Universal Robots URScript: script_ur3e.urscript

def ur3e_dibujar():
  textmsg("=== UR3e: inicio del programa ===")
  q_home = get_actual_joint_positions()
  textmsg("UR3e HOME guardado")
  # === Ir al origen calibrado: UR3e ===
  textmsg("UR3e - yendo al origen calibrado")
  x0 = -0.52777
  y0 = -0.01601
  z_mesa = 0.00821
  rx = 1.34600
  ry = 2.83900
  rz = 0.00000
  # Primero se acerca por arriba; nunca va directamente a la Z baja.
  movel(p[x0, y0, z_mesa+0.06000, rx, ry, rz], a=0.03, v=0.05)
  sleep(0.3)
  # === Detección única de superficie por fuerza: UR3e ===
  textmsg("UR3e - Detectando superficie una sola vez...")
  zero_ftsensor()
  sleep(0.5)
  i_f = 0
  while (force() < 2.000 and i_f < 2000):
    speedl([0, 0, -0.00800, 0, 0, 0], 0.25, 0.02)
    i_f = i_f + 1
  end
  stopl(3.0)
  sleep(0.2)
  if (i_f >= 2000):
    popup("UR3e: No se detectó superficie. Revisa posición inicial y F_UMBRAL.", error=True)
    halt
  end
  z_contacto = get_actual_tcp_pose()[2]
  z_dibujo = z_contacto + 0.00150
  textmsg("UR3e - z_contacto=", z_contacto)
  textmsg("UR3e - z_dibujo=", z_dibujo)
  movel(p[x0, y0, z_dibujo+0.02500, rx, ry, rz], a=0.03, v=0.04)
  sleep(0.2)
  # === Dibujo - UR3e - 3 trazos ===

  # --- Trazo 1 / 3 ---
  textmsg("UR3e - Trazo 1 de 3")
  movel(p[x0+-0.00248, y0+0.02956, z_dibujo+0.02500, rx, ry, rz], a=0.03, v=0.04)
  movel(p[x0+-0.00248, y0+0.02956, z_dibujo, rx, ry, rz], a=0.006, v=0.002)
  movel(p[x0+-0.00217, y0+0.02987, z_dibujo, rx, ry, rz], a=0.008, v=0.025, r=0.0002)
  movel(p[x0+0.00186, y0+0.02987, z_dibujo, rx, ry, rz], a=0.008, v=0.025, r=0.0002)
  movel(p[x0+0.00495, y0+0.02894, z_dibujo, rx, ry, rz], a=0.008, v=0.025, r=0.0002)
  movel(p[x0+0.00805, y0+0.02708, z_dibujo, rx, ry, rz], a=0.008, v=0.025, r=0.0002)
  movel(p[x0+0.00990, y0+0.02523, z_dibujo, rx, ry, rz], a=0.008, v=0.025, r=0.0002)
  movel(p[x0+0.01114, y0+0.02306, z_dibujo, rx, ry, rz], a=0.008, v=0.025, r=0.0002)
  movel(p[x0+0.01176, y0+0.02089, z_dibujo, rx, ry, rz], a=0.008, v=0.025, r=0.0002)
  movel(p[x0+0.01176, y0+0.01811, z_dibujo, rx, ry, rz], a=0.008, v=0.025, r=0.0002)
  movel(p[x0+0.01021, y0+0.01439, z_dibujo, rx, ry, rz], a=0.008, v=0.025, r=0.0002)
  movel(p[x0+0.00619, y0+0.00913, z_dibujo, rx, ry, rz], a=0.008, v=0.025, r=0.0002)
  movel(p[x0+0.00526, y0+0.00913, z_dibujo, rx, ry, rz], a=0.008, v=0.025, r=0.0002)
  movel(p[x0+0.00433, y0+0.00975, z_dibujo, rx, ry, rz], a=0.008, v=0.025, r=0.0002)
  movel(p[x0+0.00217, y0+0.01037, z_dibujo, rx, ry, rz], a=0.008, v=0.025, r=0.0002)
  movel(p[x0+-0.00217, y0+0.01037, z_dibujo, rx, ry, rz], a=0.008, v=0.025, r=0.0002)
  movel(p[x0+-0.00248, y0+0.01006, z_dibujo, rx, ry, rz], a=0.008, v=0.025, r=0.0002)
  movel(p[x0+-0.00464, y0+0.00975, z_dibujo, rx, ry, rz], a=0.008, v=0.025, r=0.0002)
  movel(p[x0+-0.00557, y0+0.00913, z_dibujo, rx, ry, rz], a=0.008, v=0.025, r=0.0002)
  movel(p[x0+-0.00650, y0+0.00913, z_dibujo, rx, ry, rz], a=0.008, v=0.025, r=0.0002)
  movel(p[x0+-0.01021, y0+0.01408, z_dibujo, rx, ry, rz], a=0.008, v=0.025, r=0.0002)
  movel(p[x0+-0.01145, y0+0.01625, z_dibujo, rx, ry, rz], a=0.008, v=0.025, r=0.0002)
  movel(p[x0+-0.01207, y0+0.01842, z_dibujo, rx, ry, rz], a=0.008, v=0.025, r=0.0002)
  movel(p[x0+-0.01207, y0+0.02058, z_dibujo, rx, ry, rz], a=0.008, v=0.025, r=0.0002)
  movel(p[x0+-0.01114, y0+0.02368, z_dibujo, rx, ry, rz], a=0.008, v=0.025, r=0.0002)
  movel(p[x0+-0.00990, y0+0.02554, z_dibujo, rx, ry, rz], a=0.008, v=0.025, r=0.0002)
  movel(p[x0+-0.00743, y0+0.02770, z_dibujo, rx, ry, rz], a=0.008, v=0.025, r=0.0002)
  movel(p[x0+-0.00526, y0+0.02894, z_dibujo, rx, ry, rz], a=0.008, v=0.025, r=0.0002)
  movel(p[x0+-0.00279, y0+0.02956, z_dibujo, rx, ry, rz], a=0.008, v=0.025, r=0.0002)
  movel(p[x0+-0.00279, y0+0.02956, z_dibujo+0.02500, rx, ry, rz], a=0.03, v=0.04)

  # --- Trazo 2 / 3 ---
  textmsg("UR3e - Trazo 2 de 3")
  movel(p[x0+0.01052, y0+-0.00696, z_dibujo+0.02500, rx, ry, rz], a=0.03, v=0.04)
  movel(p[x0+0.01052, y0+-0.00696, z_dibujo, rx, ry, rz], a=0.006, v=0.002)
  movel(p[x0+0.01083, y0+-0.00665, z_dibujo, rx, ry, rz], a=0.008, v=0.025, r=0.0002)
  movel(p[x0+0.01238, y0+-0.00665, z_dibujo, rx, ry, rz], a=0.008, v=0.025, r=0.0002)
  movel(p[x0+0.01640, y0+-0.00820, z_dibujo, rx, ry, rz], a=0.008, v=0.025, r=0.0002)
  movel(p[x0+0.01733, y0+-0.00820, z_dibujo, rx, ry, rz], a=0.008, v=0.025, r=0.0002)
  movel(p[x0+0.01919, y0+-0.00913, z_dibujo, rx, ry, rz], a=0.008, v=0.025, r=0.0002)
  movel(p[x0+0.02074, y0+-0.01037, z_dibujo, rx, ry, rz], a=0.008, v=0.025, r=0.0002)
  movel(p[x0+0.02229, y0+-0.01223, z_dibujo, rx, ry, rz], a=0.008, v=0.025, r=0.0002)
  movel(p[x0+0.02321, y0+-0.01408, z_dibujo, rx, ry, rz], a=0.008, v=0.025, r=0.0002)
  movel(p[x0+0.02352, y0+-0.01656, z_dibujo, rx, ry, rz], a=0.008, v=0.025, r=0.0002)
  movel(p[x0+0.02383, y0+-0.01687, z_dibujo, rx, ry, rz], a=0.008, v=0.025, r=0.0002)
  movel(p[x0+0.02321, y0+-0.02058, z_dibujo, rx, ry, rz], a=0.008, v=0.025, r=0.0002)
  movel(p[x0+0.02136, y0+-0.02399, z_dibujo, rx, ry, rz], a=0.008, v=0.025, r=0.0002)
  movel(p[x0+0.01857, y0+-0.02677, z_dibujo, rx, ry, rz], a=0.008, v=0.025, r=0.0002)
  movel(p[x0+0.01671, y0+-0.02801, z_dibujo, rx, ry, rz], a=0.008, v=0.025, r=0.0002)
  movel(p[x0+0.01207, y0+-0.02956, z_dibujo, rx, ry, rz], a=0.008, v=0.025, r=0.0002)
  movel(p[x0+0.00929, y0+-0.02956, z_dibujo, rx, ry, rz], a=0.008, v=0.025, r=0.0002)
  movel(p[x0+0.00526, y0+-0.02801, z_dibujo, rx, ry, rz], a=0.008, v=0.025, r=0.0002)
  movel(p[x0+0.00248, y0+-0.02523, z_dibujo, rx, ry, rz], a=0.008, v=0.025, r=0.0002)
  movel(p[x0+0.00093, y0+-0.02151, z_dibujo, rx, ry, rz], a=0.008, v=0.025, r=0.0002)
  movel(p[x0+0.00093, y0+-0.01377, z_dibujo, rx, ry, rz], a=0.008, v=0.025, r=0.0002)
  movel(p[x0+0.00124, y0+-0.01346, z_dibujo, rx, ry, rz], a=0.008, v=0.025, r=0.0002)
  movel(p[x0+0.00433, y0+-0.01285, z_dibujo, rx, ry, rz], a=0.008, v=0.025, r=0.0002)
  movel(p[x0+0.00712, y0+-0.01130, z_dibujo, rx, ry, rz], a=0.008, v=0.025, r=0.0002)
  movel(p[x0+0.00960, y0+-0.00882, z_dibujo, rx, ry, rz], a=0.008, v=0.025, r=0.0002)
  movel(p[x0+0.01052, y0+-0.00727, z_dibujo, rx, ry, rz], a=0.008, v=0.025, r=0.0002)
  movel(p[x0+0.01052, y0+-0.00727, z_dibujo+0.02500, rx, ry, rz], a=0.03, v=0.04)

  # --- Trazo 3 / 3 ---
  textmsg("UR3e - Trazo 3 de 3")
  movel(p[x0+-0.00186, y0+0.00820, z_dibujo+0.02500, rx, ry, rz], a=0.03, v=0.04)
  movel(p[x0+-0.00186, y0+0.00820, z_dibujo, rx, ry, rz], a=0.006, v=0.002)
  movel(p[x0+-0.00155, y0+0.00851, z_dibujo, rx, ry, rz], a=0.008, v=0.025, r=0.0002)
  movel(p[x0+0.00124, y0+0.00851, z_dibujo, rx, ry, rz], a=0.008, v=0.025, r=0.0002)
  movel(p[x0+0.00526, y0+0.00696, z_dibujo, rx, ry, rz], a=0.008, v=0.025, r=0.0002)
  movel(p[x0+0.00867, y0+0.00325, z_dibujo, rx, ry, rz], a=0.008, v=0.025, r=0.0002)
  movel(p[x0+0.00990, y0+-0.00046, z_dibujo, rx, ry, rz], a=0.008, v=0.025, r=0.0002)
  movel(p[x0+0.00960, y0+-0.00418, z_dibujo, rx, ry, rz], a=0.008, v=0.025, r=0.0002)
  movel(p[x0+0.00805, y0+-0.00727, z_dibujo, rx, ry, rz], a=0.008, v=0.025, r=0.0002)
  movel(p[x0+0.00464, y0+-0.01037, z_dibujo, rx, ry, rz], a=0.008, v=0.025, r=0.0002)
  movel(p[x0+0.00124, y0+-0.01161, z_dibujo, rx, ry, rz], a=0.008, v=0.025, r=0.0002)
  movel(p[x0+-0.00279, y0+-0.01130, z_dibujo, rx, ry, rz], a=0.008, v=0.025, r=0.0002)
  movel(p[x0+-0.00588, y0+-0.00975, z_dibujo, rx, ry, rz], a=0.008, v=0.025, r=0.0002)
  movel(p[x0+-0.00867, y0+-0.00665, z_dibujo, rx, ry, rz], a=0.008, v=0.025, r=0.0002)
  movel(p[x0+-0.00960, y0+-0.00480, z_dibujo, rx, ry, rz], a=0.008, v=0.025, r=0.0002)
  movel(p[x0+-0.00990, y0+-0.00263, z_dibujo, rx, ry, rz], a=0.008, v=0.025, r=0.0002)
  movel(p[x0+-0.01021, y0+-0.00232, z_dibujo, rx, ry, rz], a=0.008, v=0.025, r=0.0002)
  movel(p[x0+-0.00990, y0+0.00077, z_dibujo, rx, ry, rz], a=0.008, v=0.025, r=0.0002)
  movel(p[x0+-0.00836, y0+0.00418, z_dibujo, rx, ry, rz], a=0.008, v=0.025, r=0.0002)
  movel(p[x0+-0.00495, y0+0.00727, z_dibujo, rx, ry, rz], a=0.008, v=0.025, r=0.0002)
  movel(p[x0+-0.00217, y0+0.00820, z_dibujo, rx, ry, rz], a=0.008, v=0.025, r=0.0002)
  movel(p[x0+-0.00217, y0+0.00820, z_dibujo+0.02500, rx, ry, rz], a=0.03, v=0.04)

  textmsg("UR3e - Dibujo completado")
  textmsg("UR3e - Volviendo a HOME")
  movej(q_home, a=0.03, v=0.05)
  textmsg("UR3e - En HOME. Avisando al PC")
  socket_conn = socket_open("192.168.56.2", 50001, "pc_sync")
  if (not socket_conn):
    textmsg("UR3e - Error conectando con PC 192.168.56.2:50001")
    popup("UR3e no pudo conectar con el servidor Python del PC.", error=True)
    halt
  else:
    socket_send_string("LISTO", "pc_sync")
    sleep(0.2)
    socket_close("pc_sync")
    textmsg("UR3e - LISTO enviado")
  end
  textmsg("UR3e - Programa terminado")
end
ur3e_dibujar()
